# EPICS substitutions: iocBoot/iocTest/array_test.substitutions
# asyn record for the underlying asyn octet port
file "$(ASYN)/db/asynRecord.db" { pattern
{P,           R,       PORT,      ADDR,   IMAX,    OMAX}
{SIM1:    OctetAsyn,   sim1,        0,      80,      80}
}

# Address 0, UINT16 data type
file "../../db/intarray_in.template" { pattern
{P,            R,         PORT,     ADDR, NELM,        SCAN}
{SIM1:,    UINT16:Array,    UINT16,   10,  20,     "I/O Intr"}
}

file "../../db/poll_delay.template" { pattern
{P,           R,            PORT}
{SIM1:,    UINT16:PollDelay, UINT16}
}

file "../../db/poll_trigger.template" { pattern
{P,           R,            PORT}
{SIM1:,    UINT16:PollTrigger, UINT16}
}

# Address 20, INT16 data type
file "../../db/intarray_in.template" { pattern
{P,            R,           PORT,  ADDR,   NELM,        SCAN}
{SIM1:,    INT16:Array,    INT16,    10,     20,     "I/O Intr"}
}

file "../../db/poll_delay.template" { pattern
{P,            R,            PORT}
{SIM1:,    INT16:PollDelay, INT16}
}

file "../../db/poll_trigger.template" { pattern
{P,           R,            PORT}
{SIM1:,    INT16:PollTrigger, INT16}
}

# Address 40, INT32_LE data type
file "../../db/intarray_in.template" { pattern
{P,            R,            PORT,   ADDR, NELM,        SCAN}
{SIM1:,    INT32_LE:Array,  INT32_LE,  10,   20,     "I/O Intr"}
}

file "../../db/poll_delay.template" { pattern
{P,            R,            PORT}
{SIM1:,    INT32_LE:PollDelay, INT32_LE}
}

file "../../db/poll_trigger.template" { pattern
{P,           R,               PORT}
{SIM1:,    INT32_LE:PollTrigger, INT32_LE}
}

# Address 60, INT32_BE data type
file "../../db/intarray_in.template" { pattern
{P,            R,            PORT,    ADDR,  NELM,        SCAN}
{SIM1:,    INT32_BE:Array,  INT32_BE,   10,     20,     "I/O Intr"}
}

file "../../db/poll_delay.template" { pattern
{P,            R,            PORT}
{SIM1:,    INT32_BE:PollDelay, INT32_BE}
}

file "../../db/poll_trigger.template" { pattern
{P,           R,               PORT}
{SIM1:,    INT32_BE:PollTrigger, INT32_BE}
}
